PROGRAM MAIN
VAR
	a:int;
END_VAR

END_PROGRAM

(* stored: Version 1.1.0.1
   POU MAIN: Id {3cb0a3fe-7295-4bdd-b9b4-23d8f9c61c3e}, SpecialFunc None *)
